FUNCTION_BLOCK FB_KontrolleEndschalter 
VAR_INPUT
	errorOffset : WORD := 600;
END_VAR
VAR_OUTPUT
	bError : BOOL;
	nErrNo : WORD;
END_VAR
VAR
END_VAR

(* Netzwerk: 4 Kontr. Endschalter *)
(*
U "T 3" T3 -- Fehler-Kontr.Maschine (keine Bewegung)
U "T 72" T72 -- Verz. Alles OK von PNOZ
SPBN kk
*)
nErrNo := 0;
bError := FALSE;
IF NOT (GVL.tonFehlerKontrMaschine.Q AND GVL.tonSAFETYok.Q) THEN
	RETURN;
END_IF

(*
UN "A 1.7" A1.7 -- Y-10 Drahthalter+Führung zu
UN "E1_0" E1.0 -- R Drahthalter offen
S "F40 E1.0f" M104.0 -- Drahthalter nicht offen
*)
IF NOT IO.outY10DrahthaltFuehrungZU AND NOT GVL.insecDrahthalterIstOffen THEN
	GVL.errs.DrahthltNichtOffen := TRUE;
	nErrNo := errorOffset;
END_IF
(*
U "A 1.7" A1.7 -- Y-10 Drahthalter+Führung zu
U "E1_0" E1.0 -- R Drahthalter offen
S "F41 E1.0nw" M104.1 -- Drahthalter nicht zu
*)
IF IO.outY10DrahthaltFuehrungZU AND GVL.insecDrahthalterIstOffen THEN
	GVL.errs.DrahthltNichtZu := TRUE;
	nErrNo := errorOffset + 1;
END_IF


(*
UN "A 1.3" A1.3 -- Y-6 Abisolierer zu
U "E1_2" E1.2 -- N Abisolierer zu
S "F43 E1.2nw" M104.3 -- Abisolierer nicht offen
*)
IF NOT IO.outY6AbisoliererZU AND GVL.insecAbisoliererIstZU THEN
	GVL.errs.AbisolierNichtOffen := TRUE;
	nErrNo := errorOffset + 3;
END_IF


(*
U "A 1.3" A1.3 -- Y-6 Abisolierer zu
UN "E1_2" E1.2 -- N Abisolierer zu
S "F44 E1.2f" M104.4 -- Abisolierer nicht zu
*)
IF  IO.outY6AbisoliererZU AND NOT GVL.insecAbisoliererIstZU THEN
	GVL.errs.AbisolierNichtZu := TRUE;
	nErrNo := errorOffset + 4;
END_IF

(*
UN "A 1.5" A1.5 -- Y-8 Abisolierer rück
UN "E1_3" E1.3 -- R Abisolierer vorn
S "F46 E1.3f" M104.6 -- Abisolierer nicht vorn
*)
IF NOT IO.outY8AbisoliererRUECK AND NOT GVL.insecAbisoliererIstVORN THEN
	GVL.errs.AbisolierNichtVorn := TRUE;
	nErrNo := errorOffset + 6;
END_IF


(*
U "A 1.5" A1.5 -- Y-8 Abisolierer rück
UN "E1_4" E1.4 -- R Abisolierer rück (abisoliert)
S "F47 E1.4f" M104.7 -- Abisolierer nicht rück (abisoliert)
*)
IF IO.outY8AbisoliererRUECK AND NOT GVL.insecAbisoliererIstRUECK THEN
	GVL.errs.AbisolierNichtRueck := TRUE;
	nErrNo := errorOffset + 7;
END_IF


(*
U "A 1.2" A1.2 -- Y-5 Abisolierer nach links+Abdeckung zu
UN "E1_5" E1.5 -- R Abisolierer links (aus Arbeitsraum)
S "F50 E1.5f" M105.0 -- Abisolierer nicht links (aus Arbeitsraum)
*)
IF IO.outY5AbisolierNachLINKS AND NOT GVL.insecAbisoliererIstLINKS THEN
	GVL.errs.AbisolierNichtLinks := TRUE;
	nErrNo := errorOffset + 8;	
END_IF


(*
UN "A 1.2" A1.2 -- Y-5 Abisolierer nach links+Abdeckung zu
U "E1_5" E1.5 -- R Abisolierer links (aus Arbeitsraum)
S "F51 E1.5nw" M105.1 -- Abisolierer nicht rechts
*)
IF NOT IO.outY5AbisolierNachLINKS AND GVL.insecAbisoliererIstLINKS THEN
	GVL.errs.AbisolierNichtRechts := TRUE;
	nErrNo := errorOffset + 9;
END_IF


(*
U "A 1.6" A1.6 -- Y-9 Crimpen zu
UN "E1_6" E1.6 -- N Crimpzange zu
S "F53 E1.6f" M105.3 -- Crimpzange nicht zu
*)
IF IO.outY9CrimperZU AND NOT GVL.insecCrimpZangeIstZU THEN
	GVL.errs.CrimpZangeNichtZu := TRUE;
	nErrNo := errorOffset + 11;
END_IF


(*
UN "A 1.6" A1.6 -- Y-9 Crimpen zu
UN "E1_7" E1.7 -- R Crimpzange offen
S "F54 E1.7f" M105.4 -- Crimpzange nicht offen
*)
IF NOT IO.outY9CrimperZU AND NOT GVL.insecCrimpZangeIstOFFEN THEN
	GVL.errs.CrimpZangeNichtOffen := TRUE;
	nErrNo := errorOffset + 12;
END_IF


(* ToDo:
errKontaktNichtGefallen : BOOL; //(ehem. M105.5) !! nur xls File !! --
*)

//NEU
GVL.tonKontaktIstZuLangeEin(IN := GVL.insecKontaktIstGefallen, PT := T#2S);
IF GVL.tonKontaktIstZuLangeEin.Q THEN
	GVL.errs.DauerMlgKontaktGefallen := TRUE; //(ehem. 105.6) !! nur xls File !! --
	nErrNo := errorOffset + 14;
END_IF
(*
U "A 1.1" A1.1 -- Y-4 Crimpeinheit vor
UN "E2_1" E2.1 -- R Crimpeinheit vorn
S "F60 E2.1f" M106.0 -- Crimpeinheit nicht vorn
*)
IF IO.outY4CrimpEinheitVOR AND NOT GVL.insecCrimpEinheitIstVORN THEN
	GVL.errs.CrimpeinheitNichtVorn := TRUE;
nErrNo := errorOffset + 16;	
END_IF


(*
UN "A 1.1" A1.1 -- Y-4 Crimpeinheit vor
UN "E2_4" E2.4 -- R Crimpeinheit rück
S "F61 E2.4f" M106.1 -- Crimpeinheit nicht rück
*)
IF NOT IO.outY4CrimpEinheitVOR AND NOT GVL.insecCrimpEinheitIstRUECK THEN
	GVL.errs.CrimpeinheitNichtRueck := TRUE;
nErrNo := errorOffset + 17;	
END_IF


(*
U "A 1.0" A1.0 -- Y-3 Kontakt-Schieben
UN "E2_2" E2.2 -- R Kontakt-Schieben vorn
S "F62 E2.2f" M106.2 -- Kontakt-Schieben nicht vorn
*)
IF IO.outY3KontaktSchieben AND NOT GVL.insecKontaktSchiebenVORN THEN
	GVL.errs.KontaktSchiebenNichtVorn := TRUE;
	nErrNo := errorOffset + 18;
END_IF


(*
UN "A 1.0" A1.0 -- Y-3 Kontakt-Schieben
U "E2_2" E2.2 -- R Kontakt-Schieben vorn
S "F63 E2.2nw" M106.3 -- Kontakt-Schieben nicht rück
*)
IF NOT IO.outY3KontaktSchieben AND GVL.insecKontaktSchiebenVORN THEN
	GVL.errs.KontaktSchiebenNichtRueck := TRUE;
	nErrNo := errorOffset + 19;
END_IF


(*
U "A 0.6" A0.6 -- Y-1 Ausstoßen
UN "E2_3" E2.3 -- R Ausstoßen vorn
S "F64 E2.3f" M106.4 -- Ausstoßen nicht vorn
*)
IF IO.outY1Ausstossen AND NOT GVL.insecAusstossenVORN THEN
	GVL.errs.AusstossenNichtVorn := TRUE;
	nErrNo := errorOffset + 20;	
END_IF


(*
UN "A 0.6" A0.6 -- Y-1 Ausstoßen
U "E2_3" E2.3 -- R Ausstoßen vorn
S "F65 E2.3nw" M106.5 -- Ausstoßen nicht rück
*)
IF NOT IO.outY1Ausstossen AND GVL.insecAusstossenVORN THEN
	GVL.errs.AusstossenNichtRueck := TRUE;
	nErrNo := errorOffset + 21;
END_IF


//NBT-NEU
IF nErrNo <> 0 THEN
	bError := TRUE;
END_IF

(*
kk: BLD 130
*)

END_FUNCTION_BLOCK

(* stored: Version 1.1.0.1, ProductVersion 3.1.4024.3
   POU FB_KontrolleEndschalter: Id {499e0784-d2fb-4b41-b1d0-c3cfa7eddd3f}, SpecialFunc None *)
